# B&R Automation Studio project NAEUL004C00R13L518F00 (part 77)

#### Init.st
```iecst
(** 2019-03-25 **)
PROGRAM _INIT

	(* Always Change If Project Change *)

	//Physical Configuration
//	tMtrOffDlyTm	:= T#0s;

	//Pass Address To Global Address For External Use
	//Action, State & Status
	p_LifterMagConv2Stat		:= ADR(eStat);
	p_LifterMagConv2Status		:= ADR(eStatus);
	p_LifterMagConv2StatTxt		:= ADR(sStatTxt);

	//Alarm
	p_LifterMagConv2AlmData		:= ADR(tyAlmData);

	//Output
	p_LifterMagConv2HvMag				:= ADR(bHvMag);
	p_LifterMagConv2MtrSigOnOrLToR		:= ADR(bMtrSigOnOrLToR);
	p_LifterMagConv2MtrDirOrRToL		:= ADR(bMtrDirOrRToL);

	p_LifterMagConv2ClprClampCtrl	:= ADR(bClprClampCtrl);
	p_LifterMagConv2ClprTwoOutCtrl	:= ADR(bClprTwoOutputControl);

	(* Always Change If Project Change *)

END_PROGRAM
```

Listed in the project but not available here: Logical/NtLibraries/NtGeneral/NtGeneral.fun, Logical/NtLibraries/NtGeneral/fbSenFltr.st, Logical/NtLibraries/NtGeneral/fValidCharStringInChkr.st, Logical/NtLibraries/NtGeneral/fInvalidCharStringInChkr.st, Logical/NtLibraries/NtGeneral/fCheckDuplicate.st, Logical/NtLibraries/NtGeneral/fCheckExist.st, Logical/NtLibraries/NtGeneral/fStringSearch.st, Logical/NtLibraries/NtGeneral/fIPValid.st, Logical/NtLibraries/NtGeneral/fConvertUINTToHex.st, Logical/NtLibraries/NtGeneral/fConvertUSINTToHex.st, Logical/NtLibraries/NtGeneral/fConvertToLower_254.st, Logical/NtLibraries/NtUI/NtUI.fun, Logical/NtLibraries/NtUI/fUIInRtStatLock.st, Logical/NtLibraries/NtUI/fUIInRtStatHide.st, Logical/NtLibraries/NtUI/fUIInRtStatFocus.st, Logical/NtLibraries/NtUI/fUIOutRtStatCursor1Valid.st, Logical/NtLibraries/NtUI/fUIInRtStatOpenTP.st, Logical/NtLibraries/NtUI/fUIOutRtStatCursor2Valid.st, Logical/NtLibraries/NtUI/fUIOutRtStatHasFocus.st, Logical/NtLibraries/NtUI/fUIInRtStatOff.st, Logical/NtLibraries/NtUI/fUIOutRtStatInEdit.st, Logical/NtLibraries/NtUI/fUIOutRtStatOnLock.st, Logical/NtLibraries/NtUI/fUIOutRtStatTPIsOpen.st, Logical/NtLibraries/NtUI/fbTouchGetAction.st, Logical/NtLibraries/NtUI/fbTouchGetSlideDist.st, Logical/NtLibraries/NtUI/fbTouchGetTap.st, Logical/NtLibraries/NtUI/fbTableCtrl.st, Logical/NtLibraries/NtUI/fbTableCtrl_v2.st, Logical/NtLibraries/NtUI/fbTouchFilter.st, Logical/NtLibraries/NtOpConXML/Constants.var, Logical/UI/UI/Act_LinkAction.st, Logical/UI/UI/Cyclic.st, Logical/UI/UI/Act_Initial.st, Logical/UI/UI/Act_Action.st, Logical/UI/UI/Act_Main/Act_Main_C0007.st, Logical/UI/UI/Act_Main/Act_Main_P0300.st, Logical/UI/UI/Act_Background.st, Logical/UI/UI/Act_Background/Action/C0001, Logical/UI/UI/Act_Background/Action/C0002, Logical/UI/UI/Act_Background/Action/C0003, Logical/UI/UI/Act_Background/Action/C0006, Logical/UI/UI/Act_Background/Action/C0008, Logical/UI/UI/Act_Background/Action/C0010, Logical/UI/UI/Act_Background/Action/P0400/Act_OptP0400Mask.st, Logical/UI/UI/Act_Background/Action/P0400/Act_OptP0400Sort.st, Logical/UI/UI/Act_Background/Action/P0400/Act_OptP0400RcpPopUp.st, Logical/UI/UI/Act_Background/Action/P0700/Act_OptP0700Mask.st, Logical/UI/UI/Act_Background/Action/P1000/Act_ExitP1000.st, Logical/UI/UI/Act_Background/Action/P1022/Act_ExitP1022.st, Logical/UI/UI/Act_Background/Action/P1022/Act_OptP1022DisLF.st, Logical/UI/UI/Act_Background/Action/P1024/Act_ExitP1024.st, Logical/UI/UI/Act_Background/Action/P1040/Act_OptP1040RcpPopUp.st, Logical/UI/UI/Act_Background/Action/P1050/Act_OptP1050Online.st, Logical/UI/UI/Act_Background/Action/P1050/Act_OptP1050Offline.st, Logical/UI/UI/Act_Background/Action/P1050/Act_OptP1050Mask.st, Logical/UI/UI/Act_Background/Action/P1050/Act_OptP1050ShftUp.st, Logical/UI/UI/Act_Background/Action/P1050/Act_OptP1050ShftDwn.st, Logical/UI/UI/Act_Background/Action/P1080/Act_ExitP1080.st, Logical/UI/UI/Act_Background/Action/P1080/Act_OptP1080EditAccess.st, Logical/UI/UI/Act_Background/Action/P1080/Act_OptP1080AddUsr.st, Logical/UI/UI/Act_Background/Action/P1080/Act_OptP1080DelUsr.st, Logical/UI/UI/Act_Background/Action/P1080/Act_OptP1080EditUsr.st, Logical/Startup/Startup/Act_Main/Act_Main_Done.st, Logical/General/General.typ, Logical/General/General.var, Logical/General/General/Init.st, Logical/General/General/Act_InitGlobal.st, Logical/General/General/InputRef_Link.var, Logical/General/General/Act_LinkAction.st, Logical/General/General/Act_Link.st, Logical/General/General/Cyclic.st, Logical/General/General/Act_InitLocal.st, Logical/General/General/Act_Initial.st, Logical/General/General/Act_Action.st, Logical/General/General/Act_Main.st, Logical/General/General/InputRef.var, Logical/General/General/Local.var, Logical/UsrFolder/UsrFolder.var, Logical/UsrFolder/UsrFolder/Act_Initial.st, Logical/LibVer/LibVer/Init.st, Logical/LibVer/LibVer/Act_InitGlobal.st, Logical/LibVer/LibVer/InputRef_Link.var, Logical/LibVer/LibVer/Act_LinkAction.st, Logical/LibVer/LibVer/Act_Link.st, Logical/LibVer/LibVer/Act_RstErr.st, Logical/LibVer/LibVer/Act_InitLocal.st, Logical/LibVer/LibVer/Act_Action.st, Logical/LibVer/LibVer/InputRef.var, Logical/LibVer/LibVer/Local.var, Logical/Time/Time/Act_InitGlobal.st, Logical/Time/Time/InputRef_Link.var, Logical/Time/Time/Act_LinkAction.st, Logical/Time/Time/Act_Link.st, Logical/Time/Time/Act_RstErr.st, Logical/Time/Time/Act_InitLocal.st, Logical/Time/Time/Act_Action.st, Logical/Time/Time/Act_Background.st, Logical/Time/Time/Act_CombineErr.st, Logical/Time/Time/InputRef.var, Logical/TLBuz/TLBuz/Act_Initial.st, Logical/Alarm/Alarm/Act_LinkAction.st, Logical/Alarm/Alarm/Act_RstErr.st, Logical/Alarm/Alarm/Act_InitLocal.st, Logical/Alarm/Alarm/Act_Action.st, Logical/Alarm/Alarm/Act_Background.st, Logical/ProdRcp/ProdRcp/InputRef.var, Logical/UsrMgmt/UsrMgmt.var, Logical/OvenInfo/OvenInfoA/Act_LinkEn.st, Logical/OvenInfo/OvenInfoA/Act_InitLocal.st, Logical/OvenInfo/OvenInfoA/Act_Action.st, Logical/OvenInfo/OvenInfoA/Act_Background.st, Logical/Buffer/Buffer2/Act_RstErr.st, Logical/Buffer/Buffer2/Act_InitLocal.st, Logical/Buffer/Buffer2/Act_Background.st, Logical/Buffer/Buffer2/InputRef.var, Logical/Buffer/Buffer2/Local.var, Logical/Buffer/Buffer3/Act_RstErr.st, Logical/Buffer/Buffer3/Act_InitLocal.st, Logical/Buffer/Buffer3/Act_Action.st, Logical/Buffer/Buffer3/Act_Main.st, Logical/Buffer/Buffer3/Act_Background.st, Logical/Buffer/BufferMagB/Cyclic.st, Logical/Buffer/BufferMagB/Act_Initial.st, Logical/Pneu/PneuOutShutter2/Cyclic.st, Logical/Pneu/PneuOutShutter2/Act_Initial.st, Logical/Pneu/PneuOutShutter2/Act_Main.st, Logical/Pneu/PneuOutShutter2/Act_Alarm.st, Logical/Pneu/PneuOutShutter2/Local.var, Logical/Pneu/PneuNoSenStopperB/InputRef_Link.var, Logical/Pneu/PneuNoSenStopperB/Act_LinkEn.st, Logical/Pneu/PneuNoSenStopperB/Act_Link.st, Logical/Pneu/PneuNoSenStopperB/Cyclic.st, Logical/Pneu/PneuNoSenStopperB/Act_RstErr.st, Logical/Pneu/PneuNoSenStopperB/Act_InitLocal.st, Logical/Pneu/PneuNoSenStopperB/Act_Initial.st, Logical/Pneu/PneuNoSenStopperB/Act_Action.st, Logical/Pneu/PneuNoSenStopperB/Act_Main.st, Logical/Pneu/PneuNoSenStopperB/InputRef.var, Logical/Pneu/PneuNoSenStopperB/Local.var, Logical/MagConv_LiftnTrav/MagConv2Clp1/Act_LinkEn.st, Logical/MagConv_LiftnTrav/MagConv2Clp1/Cyclic.st, Logical/MagConv_LiftnTrav/MagConv2Clp1/Act_RstErr.st, Logical/MagConv_LiftnTrav/MagConv2Clp1/Act_InitLocal.st, Logical/MagConv_LiftnTrav/MagConv2Clp1/Act_Alarm.st, Logical/MagConv_LiftnTrav/MagConv2Clp3/InputRef_Link.var, Logical/MagConv_LiftnTrav/MagConv2Clp3/Act_RstErr.st, Logical/MagConv_LiftnTrav/MagConv2Clp3/Act_Action.st, Logical/MagConv_LiftnTrav/MagConv2Clp3/InputRef.var, Logical/SOT/DSSOT3/Act_InputConfig.st, Logical/SOT/DSSOT3/Act_Initial.st, Logical/SOT/DSSOT3/Act_Main.st, Logical/SOT/DSSOT3/Act_Background.st, Logical/LF/LFLeader/InputRef_Link.var, Logical/LF/LFLeader/Cyclic.st, Logical/LF/Follower2/Cyclic.st, Logical/LF/Follower2/Act_RstErr.st, Logical/LF/Follower2/Act_Initial.st, Logical/LF/Follower2/Act_Background_UpdtData.st, Logical/Machine/Machine/Act_Initial.st, Logical/AGVCom/AGV/Act_Background.st, Logical/AGVCom/AGV3/Act_Background.st, Logical/CANOpenServo/CANOpenServo.typ, Logical/CANOpenServo/AW/AWOpen.var, Logical/CANOpenServo/AW/AWOpen/Act_LinkEn.st, Logical/CANOpenServo/AW/AWOpen/Cyclic.st, Logical/CANOpenServo/AW/AWOpen/Act_RstErr.st, Logical/CANOpenServo/AW/AWOpen/Act_Action.st, Logical/CANOpenServo/AW/AWOpen/Act_Main.st, Logical/CANOpenServo/AW/AWOpen/Act_Main_Disable.st, Logical/CANOpenServo/AW/AWOpen/Act_CombineErr.st, Logical/CANOpenServo/AW/AWPushOrPuller/Act_LinkEn.st, Logical/CANOpenServo/AW/AWPushOrPuller/Cyclic.st, Logical/CANOpenServo/AW/AWPushOrPuller/Act_RstErr.st, Logical/CANOpenServo/AW/AWPushOrPuller/Act_InitLocal.st, Logical/CANOpenServo/AW/AWPushOrPuller/Act_Action.st, Logical/CANOpenServo/AW/AWPushOrPuller/Act_Main_Disable.st, Logical/CANOpenServo/AW/AWPushOrPuller/Act_CombineErr.st, Logical/CANOpenServo/Trav/Trav/Act_LinkEn.st, Logical/CANOpenServo/Trav/Trav/Act_RstErr.st, Logical/CANOpenServo/Trav/Trav/Act_CombineErr.st, Logical/CANOpenServo/Lifter/LifterBtm/Act_LinkEn.st, Logical/CANOpenServo/Lifter/LifterBtm/Cyclic.st, Logical/CANOpenServo/Lifter/LifterBtm/Act_RstErr.st, Logical/CANOpenServo/Lifter/LifterBtm/Act_Initial.st, Logical/CANOpenServo/Lifter/LifterBtm/Act_Action.st, Logical/CANOpenServo/Lifter/LifterBtm/Act_CombineErr.st, Logical/CANOpenServo/MagAW/MagAWOpen2/InputRef_Link.var, Logical/CANOpenServo/MagAW/MagAWOpen2/Act_LinkEn.st, Logical/CANOpenServo/MagAW/MagAWOpen2/Act_InitLocal.st, Logical/CANOpenServo/MagAW/MagAWOpen2/Act_RstErr.st, Logical/CANOpenServo/MagAW/MagAWOpen2/Act_Initial.st, Logical/CANOpenServo/MagAW/MagAWOpen2/Act_Action.st, Logical/CANOpenServo/MagAW/MagAWOpen2/Act_Main.st, Logical/CANOpenServo/MagAW/MagAWOpen2/Act_CombineErr.st, Logical/CANOpenServo/MagAW/MagAWOpen2/Act_Alarm.st, Logical/CANOpenServo/MagAW/MagAWOpen2/Act_Alarm3.st, Logical/CANOpenServo/MagAW/MagAWOpen2/Local.var, Logical/DOutput/DOutput/Init.st, Logical/DOutput/DOutput/Act_LinkAction.st, Logical/DOutput/DOutput/Act_Initial.st, Logical/DOutput/DOutput/Act_Action.st, Logical/Hermes/Hermes/Act_LinkEn.st, Logical/Hermes/Hermes/Act_RstErr.st, Logical/Hermes/USHermesB/Act_LinkEn.st, Logical/Hermes/USHermesB/Act_RstErr.st, Logical/Hermes/USHermesB/Act_Action.st, Logical/Hermes/USHermesB/Act_Main.st, Logical/Hermes/USHermesB/Act_Background_NotificationRcv.st, Logical/Hermes/USHermesB/Act_Background_CmpParamRcv.st, Logical/Hermes/USHermesB/Act_Background_ChkAlive.st, Logical/Hermes/USHermesB/Act_Background_ChkAliveSendPing.st, Logical/Hermes/USHermesB/Act_Background_ChkAliveRcvPing.st, Logical/Hermes/USHermesB/Act_Background_NotificationSnd.st, Logical/Hermes/USHermesB/Act_Background_Err.st, Logical/Hermes/USHermesB/Act_Main_Disable.st, Logical/Hermes/USHermesB/Act_Alarm2.st, Logical/Hermes/USHermesB/Act_Alarm4.st, Logical/LCS/LCS/Act_LinkEn.st, Logical/LCS/LCS/Cyclic.st, Logical/LCS/LCS/Act_InitLocal.st, Logical/LCS/LCS/Act_Initial.st, Logical/LCS/LCS/Act_Background.st, Logical/LCS/LCS/Act_Main_Disable.st, Logical/LCS/LCSLF.var, Logical/LCS/LCSLF/Init.st, Logical/LCS/LCSLF/Act_LinkAction.st, Logical/LCS/LCSLF/Act_Link.st, Logical/LCS/LCSLF/Cyclic.st, Logical/LCS/LCSLF/Act_RstErr.st, Logical/LCS/LCSLF/Act_InitLocal.st, Logical/LCS/LCSLF/Act_Initial.st, Logical/LCS/LCSLF/Act_Action.st, Logical/LCS/LCSLF/Act_Background.st, Logical/LCS/LCSLF/Act_Main_Disable.st, Logical/LCS/LCSLF/Act_Alarm.st, Logical/LCS/LCSLF/Local.var, Logical/Operations/Operations.typ, Logical/Operations/OpsTravLifUL/Cyclic.st, Logical/Operations/OpsTravLifUL/Act_RstErr.st, Logical/Operations/OpsTravLifUL/Act_Initial.st, Logical/Operations/OpsTravLifUL/Act_Background.st, Logical/Operations/OpsTravLifUL/Sequence/Act_LogStep.st, Logical/Operations/MagConv_StationaryPlat/OpsMagConvUL2/Cyclic.st, Logical/Operations/MagConv_StationaryPlat/OpsMagConvUL2/Act_RstErr.st, Logical/Operations/MagConv_StationaryPlat/OpsMagConvUL2/Act_AlarmInfo1.st, Logical/Operations/MagConv_StationaryPlat/OpsMagConvUL3/Sequence/Act_LogStep.st, Logical/Operations/OpsPosAllwGo/InputRef_Link.var, Logical/Operations/OpsPosAllwGo/Act_LinkEn.st, Logical/Operations/OpsPosAllwGo/Cyclic.st, Logical/Operations/OpsPosAllwGo/Act_RstErr.st, Logical/Operations/OpsPosAllwGo/Act_Initial.st, Logical/Operations/OpsPosAllwGo/Act_Background.st, Logical/Operations/OpsPosAllwGo/Act_Alarm.st, Logical/Simulation/Simulation.typ, Logical/Simulation/Simu/Init.st, Logical/Simulation/Simu/Act_LinkAction.st, Logical/Simulation/Simu/Cyclic.st, Logical/Simulation/Simu/Act_RstErr.st, Logical/Simulation/Simu/Act_InitLocal.st, Logical/Simulation/Simu/Act_Initial.st, Logical/Simulation/Simu/Act_Action.st, Logical/Simulation/Simu/Act_Main.st, Logical/Simulation/Simu/InputRef.var, Logical/OpCon/OpCon/Act_LinkEn.st, Logical/OpCon/OpCon/Act_RstErr.st, Logical/AutoRcp/AutoRcp/Act_RstErr.st
